FUNCTION_BLOCK Mo20_St80_cleaning_and_empty_check_1
(*--------------------------------------------------------------------------------------
Preh IMA Automation Amberg GmbH

<DESC>
=INSERT DESCRIPTION FROM WORKFLOWPLAN=
</DESC>


<CHANGES>
At every change add date, version´s number, abbr. of name and describe change!

Date 		|	Version	|	Author	|	change description		
--------------------------------------------------------------------------------
2017-11-23	|	1.00	|	DWO		|	initial version

</CHANGES>
<VERSION>
1.00
</VERSION>

<DEPENDENCIES>
;
</DEPENDENCIES>



 -- overview of areas for steps --
Steps [000..099]: 	Whatever Block
Steps [100..199]:	Next Whatever Block

  
----------------------------------------------------------------------------------------*)



(* _____________________ *)
(* -- Standard-Inputs -- *)
VAR_INPUT
	OrderNr: 			INT :=1;		(* Nr. Actorder *)
	MoNr: 				INT:= 20;		(* Module-Number *)
	StNr: 				INT:= 80;		(* Stationsnumber *)
	BedienEinheit: 		ZENTR_DATA;		(* Central *)
	FaultID: 			BYTE := 0;		(* ID for Error Array *)
	DisplayNr: 			INT := 1;		(* Number of Textdisplay *)
	MPart: 				INT := 1;		(* Machinepart *)
	in_InitChainTxt:	STRING(39);		(* String for Step Chain Diagnosis *)
	in_sKebaKurz:		STRING(gcKebaStKurzLen) := '1234567890'; (* optional - can also be assigned in initialisation paragraph *)
	in_sKebaBez:		STRING(gcKebaStBezLen) 	:= '11111111112222222222333333333344444444445555555555'; (* optional - can also be assigned in initialisation paragraph *)
END_VAR


(* __________________ *)
(* -- RT-Interface -- *)
VAR_INPUT
	RtNr:				INT := 01;
	RtStNr:				SINT := 08;
	RtStartimpuls:		BOOL:=FALSE;	
END_VAR

VAR_IN_OUT
	//io_RtRegister:		ARRAY[1..8] OF ARRAY[1..2] OF DataTeil; // info for all parts within roundtable - the part for the station is accessed at [RtStNr]
	io_RtStarts:		DWORD; // bit array (dword) representing station is working on roundtable (flow based)
	io_RtFreigabe:		DWORD; // bit array (dword) representing station is giving permission for table to move (state based)
	io_RtFault:			DWORD; // bit array (dword) representing error at RtStNr of roundtable
	io_RtWaiting:		DWORD; // bit array (dword) representing waiting at RtStNr of roundtable
	io_RtWarning:		DWORD; // bit array (dword) representing warning at RtStNr of roundtable
END_VAR



(* ________________________ *)
(* -- Standard-Variables -- *)
VAR PERSISTENT
	SWI: 				BOOL := FALSE;	(* Impulse step is changing forward *)
	SWR:				BOOL := FALSE;	(* Impulse step is changing backwards *)
	Schritt: 			INT := 0;		(* Current step *)
	UZ: 				TON;			(* watchtime *)
	Fault: 				BOOL;			(* Stations Error *)
	Waiting:			BOOL;			(* Station Waiting *)
	Warning:			BOOL;			(* Station Warning *)
	Betrieb: 			BOOL;			(* Enable Steps *)
	StatEin: 			BOOL;			(* Station on *)
	AllInPos: 			BOOL;			(* all cylinders in position and not actuated manually *)
	Active:				BOOL;			(* stepchain is marked as active *)
	Transport:			BOOL;			(* manual transport is enabled *)
	InitRun:			BOOL;			(* goto homepos is enabled *)
	CycleRun:			BOOL;			(* mode for single cycle is enabled *)
	ManualRun:			BOOL;			(* move cylinders manually is enabled *)
	BackwardsRun:		BOOL;			(* backwards run is enabled *)
	tonSeitSwi:			TON;			(* time since last change of step *)
	tonSeitAllInPos:	TON;			(* time since AllInPos has become TRUE *)
	i:					INT;			(* index-runner for loops *)
	j:					INT;			(* index-runner for loops *)
	xx:					FB_StepTracker;	(* auto record steps *)
	StatString:			STRING(10);		(* '+MM=SS' *)
	StartCondition:		BOOL;			(* condition for starting station *)
	bStart:				BOOL;			(* station's work on roundtable is running *)
	NestNr:				INT;			(* number of nest within fixation *)
END_VAR

VAR CONSTANT	
NEST1 :				INT :=1;
NEST2 :				INT :=2;
END_VAR

(* ___________________ *)
(* -- Error-Array 1 -- *)
VAR
	Errors1: ARRAY[1..ErrMaxBits] OF ERRDAT := [
	(* Error 01 *)		(Prio := ErrZyl, Nr:= 196, Txt:='=080-BG2 '),
	(* Error 02 *)		(Prio := ErrZyl, Nr:= 196, Txt:='=080-BG3 '),
	(* Error 03 *)		(Prio := ErrZyl, Nr:= 510, Txt:='/03 '),
	(* Error 04 *)		(Prio := ErrZyl, Nr:= 510, Txt:='/04 '),
	(* Error 05 *)		(Prio := ErrZyl, Nr:= 510, Txt:='/05            '),
	(* Error 06 *)		(Prio := ErrZyl, Nr:= 2551, Txt:='dynamic text '),
	(* Error 07 *)		(Prio := ErrZyl, Nr:= 510, Txt:='/07            '),
	(* Error 08 *)		(Prio := ErrZyl, Nr:= 510, Txt:='/08            '),
	(* Error 09 *)		(Prio := ErrZyl, Nr:= 510, Txt:='/09            '),
	(* Error 10 *)		(Prio := ErrZyl, Nr:= 510, Txt:='/10            '),
	(* Error 11 *)		(Prio := ErrZyl, Nr:= 510, Txt:='/11            '),
	(* Error 12 *)		(Prio := ErrZyl, Nr:= 510, Txt:='/12            '),
	(* Error 13 *)		(Prio := ErrZyl, Nr:= 510, Txt:='/13            '),
	(* Error 14 *)		(Prio := ErrZyl, Nr:= 510, Txt:='/14            '),
	(* Error 15 *)		(Prio := ErrZyl, Nr:= 510, Txt:='/15            '),
	(* Error 16 *)		(Prio := ErrZyl, Nr:= 510, Txt:='/16            ')];
	f1: ARRAY [1..ErrMaxBits] OF BOOL := [ErrMaxBits(FALSE)];
	Fehler1: ERRORANZ;
END_VAR

VAR CONSTANT
(* -- Error-EmptyCheck -- *)
feEmptyCheck						: ARRAY[1..2] OF INT :=[1,2];

feWaitForTaifunAtCorrectSpeed		: INT := 6;
END_VAR


(* _____________________ *)
(* -- Local Variables -- *)
VAR PERSISTENT

(* == Valve == *)
ValveTaifun					:ZYL0; (* MM1 *)

(* == Escherich Taifun == *)
ton_1s						:TON;
ton_impuls					:TON;
BDE_diTaifunUL_SpeedRpm		:DINT :=0;
BDE_diTaifunLL_SpeedRpm		:DINT :=0;

ixTaifunRotorSensor			:BOOL :=FALSE;   //=080-BG1
rtTaifunRotorSensor			:R_TRIG;

_diCurrentMotorCounts		:DINT :=0;
_arr_diSpeedMotorPerSecond	:ARRAY[1..3] OF DINT;
_diSpeedMotorPerMinuteMw	:DINT;

(* == EmptyCheck == *)
ixEmptyCheckCavity			:ARRAY[1..2] OF BOOL :=[FALSE,FALSE];
bAllCavitiesEmpty			: BOOL :=FALSE;




END_VAR




(* _____________________ *)
(* -- Function Blocks -- *)
VAR
END_VAR

(* ____________________ *)
(* -- Initialisation -- *)
IF neustart OR g_bOnlineChange THEN
	StatString 		:= RIGHT(CONCAT( '000',INT_TO_STRING(StNr) ),3); (* three digits station's prefix is being created automatically for station *)
	in_InitChainTxt := CONCAT( StatString, ' §Clean§ §Carrier§ / §Empty Check§' );
	in_sKebaKurz	:= CONCAT( StatString, ' Empty'); // 3+7 digits
	in_sKebaBez		:= in_InitChainTxt;
END_IF


KebaInitStation(
	Panelnummer		:= gKebaAktPanel,
	Aktiv			:= TRUE,
	Kurzbezeichnung	:= in_sKebaKurz,
	Bezeichnung		:= in_sKebaBez,
	ManuellAktiv	:= TRUE,
	RueckwaertsAktiv:= FALSE,
	GsAktiv			:= FALSE,
);


(* _______________________________________ *)
(* -- Entry for Step Sequence Diagnosis -- *)
InitChain(
	Step 			:= Schritt,
	InitialState 	:= TRUE,
	Fault 			:= Fault,
	Waiting 		:= Waiting,
	Warning 		:= Warning,
	AllInPos 		:= AllInPos,
	RunOpenDoor 	:= TRUE,
	Txt 			:= in_InitChainTxt,
	BedienEinheit 	:= BedienEinheit,
	Active 			:= Active,
	Transport 		:= Transport,
	InitRun 		:= InitRun,
	CycleRun 		:= CycleRun,
	ManualRun 		:= ManualRun,
	BackwardsRun 	:= BackwardsRun);
InitRun := FALSE;


(* _______________ *)
(* -- Parameter -- *)
StatEin 	:= ActOrd[MPart].ord_stat[OrderNr].sd_ein;
BDE_diTaifunUL_SpeedRpm	:= ActOrd[MPart].ord_stat[OrderNr].sd_p1;
BDE_diTaifunLL_SpeedRpm	:= ActOrd[MPart].ord_stat[OrderNr].sd_p2;


(* ____________ *)
(* -- Inputs -- *)
ixTaifunRotorSensor			:=_080_M20_MP1_BG1;

ixEmptyCheckCavity[NEST1]	:=_080_M20_MP1_BG2;
ixEmptyCheckCavity[NEST2]	:=_080_M20_MP1_BG3;


(* _______________________ *)
(* -- Timer / Watchdogs -- *)
UZ( IN:= NOT SWI AND BedienEinheit.grundbed, PT:= T#5s );
tonSeitSwi( IN := NOT SWI AND Bedieneinheit.grundbed, PT := t#30d );
tonSeitAllInPos( IN := AllInPos AND Bedieneinheit.grundbed, PT := t#30d );


(* _______________ *)
(* -- Cylinders -- *)
ValveTaifun(
	on:= , 
	enable_man:= Bedieneinheit.ventile_ok, 
	FNrMan		:=2550,
	on_vz		:= T#4S,  
	off_vz		:= T#0S, 
	FAnz		:= DisplayNr,
	StNr		:= StatString,
	ZylNr		:= '1', 
	txtVentil	:= 'MZ1', 
	ID			:= FaultID, 
	Bild		:= picStandardSchalterAus, 
	BildB		:= picStandardSchalterEin,
);

AllInPos :=	ValveTaifun.pos;

(* count motor pulses *)
rtTaifunRotorSensor( CLK := ixTaifunRotorSensor );
IF rtTaifunRotorSensor.Q THEN
	_diCurrentMotorCounts := _diCurrentMotorCounts + 1;
END_IF

ton_1s( IN := NOT ton_1s.Q AND valveTaifun.y, PT := T#1S ); // start to count pulses with valve on
IF ton_1s.Q 
THEN
	(* shift past 3 seconds in shiftregister *)
	_arr_diSpeedMotorPerSecond[3] 	:= _arr_diSpeedMotorPerSecond[2];
	_arr_diSpeedMotorPerSecond[2] 	:= _arr_diSpeedMotorPerSecond[1];
	_arr_diSpeedMotorPerSecond[1] 	:= _diCurrentMotorCounts; (* save counts of the last second to "speed per second" at [1] *) 
	_diCurrentMotorCounts 			:= 0; (* reset temporary counts *)

	(* calculate rpm by adding pulses of past 3 sec. * 20 = 60 sec. (=> result = rpm / minute) *) 
	_diSpeedMotorPerMinuteMw		:=
		(	_arr_diSpeedMotorPerSecond[1]
		+ 	_arr_diSpeedMotorPerSecond[2]
		+ 	_arr_diSpeedMotorPerSecond[3]
		)
		*	20 /2 (* / 2 Pulses per Round *); 
	
END_IF

(* __________________ *)
(* -- EmptyCheck all cavities-- *)
bAllCavitiesEmpty		:= NOT (ixEmptyCheckCavity[NEST1]
							OR 	ixEmptyCheckCavity[NEST2]);

(* __________________ *)
(* -- Treat Errors -- *)
Fehler1( ID:= FaultID, FAnz:= DisplayNr, EF:= Errors1, F:= f1 );

Fault	:= ValveTaifun.err	(* Error´s of function blocks *);
Warning := FALSE;
Waiting := FALSE;
FOR i := 1 TO ErrMaxBits BY 1 DO
	IF f1[i] THEN
		IF 		Errors1[i].Prio <= ErrZyl 			THEN Fault := TRUE;
		ELSIF	Errors1[i].Prio <= ErrEndl 			THEN Waiting := TRUE; f1[i] := FALSE;
		ELSIF	Errors1[i].Prio <= ErrWechselpos	THEN Warning := TRUE; f1[i] := FALSE; END_IF
	END_IF
END_FOR


// report Error, Waiting and Warning to cell
IF Fault 	THEN io_RtFault 	:= SETBIT32( io_RtFault,   RtStNr ); END_IF
IF Waiting 	THEN io_RtWaiting 	:= SETBIT32( io_RtWaiting, RtStNr ); END_IF
IF Warning	THEN io_RtWarning	:= SETBIT32( io_RtWarning, RtStNr ); END_IF


(* Create Errrors / Misc. Errors *)


(* __________________________________ *)
(* -- Station - Allowed to Operate -- *)
Betrieb := 	Bedieneinheit.betrieb
		AND NOT Fault
		AND NOT ManualRun
		AND BedienEinheit.ventile_ok;


(* ____________________ *)
(* -- Start Station  -- *)
IF 	RtStartimpuls THEN
	StartCondition 
		:= 	StatEin;
					
	IF StartCondition THEN bStart := TRUE; END_IF
END_IF


(* ________________ *)
(* -- Step-Chain -- *)
xx( iStep := Schritt );

(* reset flags *)
SWI := FALSE;

CASE Schritt OF
0:	xx.x := 'in basepos. - wait for prework or station´s start';
	IF  AllInPos
	AND bStart
	AND BedienEinheit.anl_ein
	AND Betrieb THEN
		Schritt := Schritt + 10;
		SWI := TRUE;
	END_IF


10:	xx.x := 'empty checking';
	IF 	AllInPos
	AND Betrieb THEN
		IF NOT bAllCavitiesEmpty THEN
			//f1[feEmptyCheck] :=TRUE;
			FOR j :=1 TO NEST2  BY  1 DO
				f1[feEmptyCheck[i]] :=ixEmptyCheckCavity[i];
			END_FOR
			
		ELSIF   	bAllCavitiesEmpty 
				AND NOT (f1[feEmptyCheck[NEST1]] 
						OR f1[feEmptyCheck[NEST2]]
						)

		THEN
		Schritt := Schritt + 10;
		SWI := TRUE;	
		END_IF
		
	END_IF

20:	xx.x := 'ionization unit is ON';	
	g_bCentralCleaningRequestOn := TRUE;						//reset request after process
	IF 	AllInPos
	AND Betrieb 
	AND g_bCentralCleaningRunning 
	THEN
		Schritt := Schritt + 10;
		SWI := TRUE;
	END_IF
	
	
30:xx.x := 'Enable valve of Taifun)';
	g_bCentralCleaningRequestOn := TRUE;
	IF	NOT Statein
		THEN
			bstart :=FALSE;
			schritt :=0;
			SWI :=TRUE;
		ELSIF AllInPos
			THEN 
				IF (_diSpeedMotorPerMinuteMw >=BDE_diTaifunLL_SpeedRpm) AND (_diSpeedMotorPerMinuteMw <=BDE_diTaifunUL_SpeedRpm)
					THEN 
						bstart :=FALSE;
						schritt :=0;
						SWI :=TRUE;
					ELSE 
						(*MV,2551,*** warte bis Taifun (Dr.Escherich) Drehzahl erreicht   
                          MV,2551,aktuell: **** rpm (von **** bis **** rpm)*)
						Errors1[feWaitForTaifunAtCorrectSpeed].Txt		:=Statstring;
						Errors1[feWaitForTaifunAtCorrectSpeed].Txt		:=concat (Errors1[feWaitForTaifunAtCorrectSpeed].Txt,
																				  RIGHT(concat(' ',DINT_TO_STRING(_diSpeedMotorPerMinuteMw)),4));
						Errors1[feWaitForTaifunAtCorrectSpeed].Txt		:=concat (Errors1[feWaitForTaifunAtCorrectSpeed].Txt,
																				  LEFT(concat(DINT_TO_STRING(BDE_diTaifunLL_SpeedRpm),' '),4));
						Errors1[feWaitForTaifunAtCorrectSpeed].Txt		:=concat (Errors1[feWaitForTaifunAtCorrectSpeed].Txt,
																				  RIGHT(concat(' ',DINT_TO_STRING(BDE_diTaifunUL_SpeedRpm)),4));
						f1[feWaitForTaifunAtCorrectSpeed]	:=TRUE;
				END_IF
	END_IF
END_CASE


(* ____________________ *)
(* -- React to Steps -- *)
IF NOT ManualRun THEN
	//turn on the ionization unit:= 	(schritt :=20)
	ValveTaifun.on := 	(schritt =30);
END_IF


(* _____________________________________ *)
(* -- Stop Roundtable Condition-Based -- *)
IF FALSE (* <----insert condition for stop here - i.e. zylVertical.y OR NOT zylVertical.a *) THEN 
	F_ResetFrgRtWithText(TRUE, RtNr, RtStNr, '010MM2 §Vertical§ §not§ §in§ §base-pos.§', io_RtFreigabe);
END_IF


(* ______________________________________ *)
(* -- Report Station is working on RT  -- *)
io_RtStarts := CSETBIT32(io_RtStarts, RtStNr, bStart);


(* _________________ *)
(* -- Set outputs -- *)

IF ManualRun THEN (* assign cylinderoutputs .y (by "AND Bedieneinheit.ventile_ok") *)
	_080_M20_MP1_QM1_MB1         	:=		ValveTaifun.y AND Bedieneinheit.ventile_ok;
	_080_M20_MP1_QM1_MB2         	:=	not ValveTaifun.y AND Bedieneinheit.ventile_ok;
ELSE (* assign cylinderoutputs .on (by "AND Bedieneinheit.ventile_ok") *)
	_080_M20_MP1_QM1_MB1         	:=		ValveTaifun.on AND Bedieneinheit.ventile_ok;
	_080_M20_MP1_QM1_MB2         	:=	not ValveTaifun.on AND Bedieneinheit.ventile_ok;
END_IF

END_FUNCTION_BLOCK

(* stored: Version 1.1.0.1, ProductVersion 3.1.4022.16
   POU Mo20_St80_cleaning_and_empty_check_1: Id {88879a90-d31f-4160-aa11-33ff87e37061}, SpecialFunc None *)
